// TIA Portal V17 export
// export: Created 2025-07-01T09:58:41.890921Z, ExportSetting WithDefaults, DisplayName Totally Integrated Automation Portal, DisplayVersion V17 Update 8, DisplayName TIA Portal Openness, DisplayVersion V17 Update 8, DisplayName TIA Portal Version Control Interface, DisplayVersion V17, DisplayName SINAMICS Startdrive Advanced, DisplayVersion V17 SP2, DisplayName SINAMICS Startdrive G110M, G120, G120C, G120D, G120P, G115D, DisplayVersion V17 SP2, DisplayName SINAMICS Startdrive G130, G150, S120, S150, SINAMICS MV, S210, DisplayVersion V17 SP2, DisplayName STEP 7 Professional, DisplayVersion V17 Update 8, DisplayName SINUMERIK ONE STEP 7 Toolbox, DisplayVersion V17 Update 12, DisplayName SINUMERIK ONE PLC Basic Program Plus, DisplayVersion V17 Update 12, DisplayName SINUMERIK 840D sl STEP 7 Toolbox, DisplayVersion V17 Update 12, DisplayName STEP 7 Safety, DisplayVersion V17 Update 6, DisplayName WinCC Advanced, DisplayVersion V17 Update 8
FUNCTION "FC442_MACHINE_RUN_OUT_ALARM_DECODING" : Void   // FC442, LAD
{ S7_Optimized_Access := 'FALSE' }
AUTHOR : ETXETAR
VERSION : 1.0
// stored: AutoNumber false, IsIECCheckEnabled false, SetENOAutomatically false, UDAEnableTagReadback false
   VAR_TEMP
      RST_ALARMS_1 : Bool;   // RESET ALARMS 1
      RST_ALARMS_2 : Bool;   // RESET ALARMS 2
      ZERO : Int;   // ZERO
      RET_VAL_1 : Int;   // RET VALUE
   END_VAR
   VAR CONSTANT
      FC_CONSTANT : Int := 440;
   END_VAR
   VAR_TEMP   // added for the SCL form of the ladder/FBD networks
      _w1 : Bool;
      _w2 : Bool;
      _w3 : Bool;
      _w4 : Bool;
      _w5 : Bool;
   END_VAR
BEGIN

REGION Network 1: ZERO
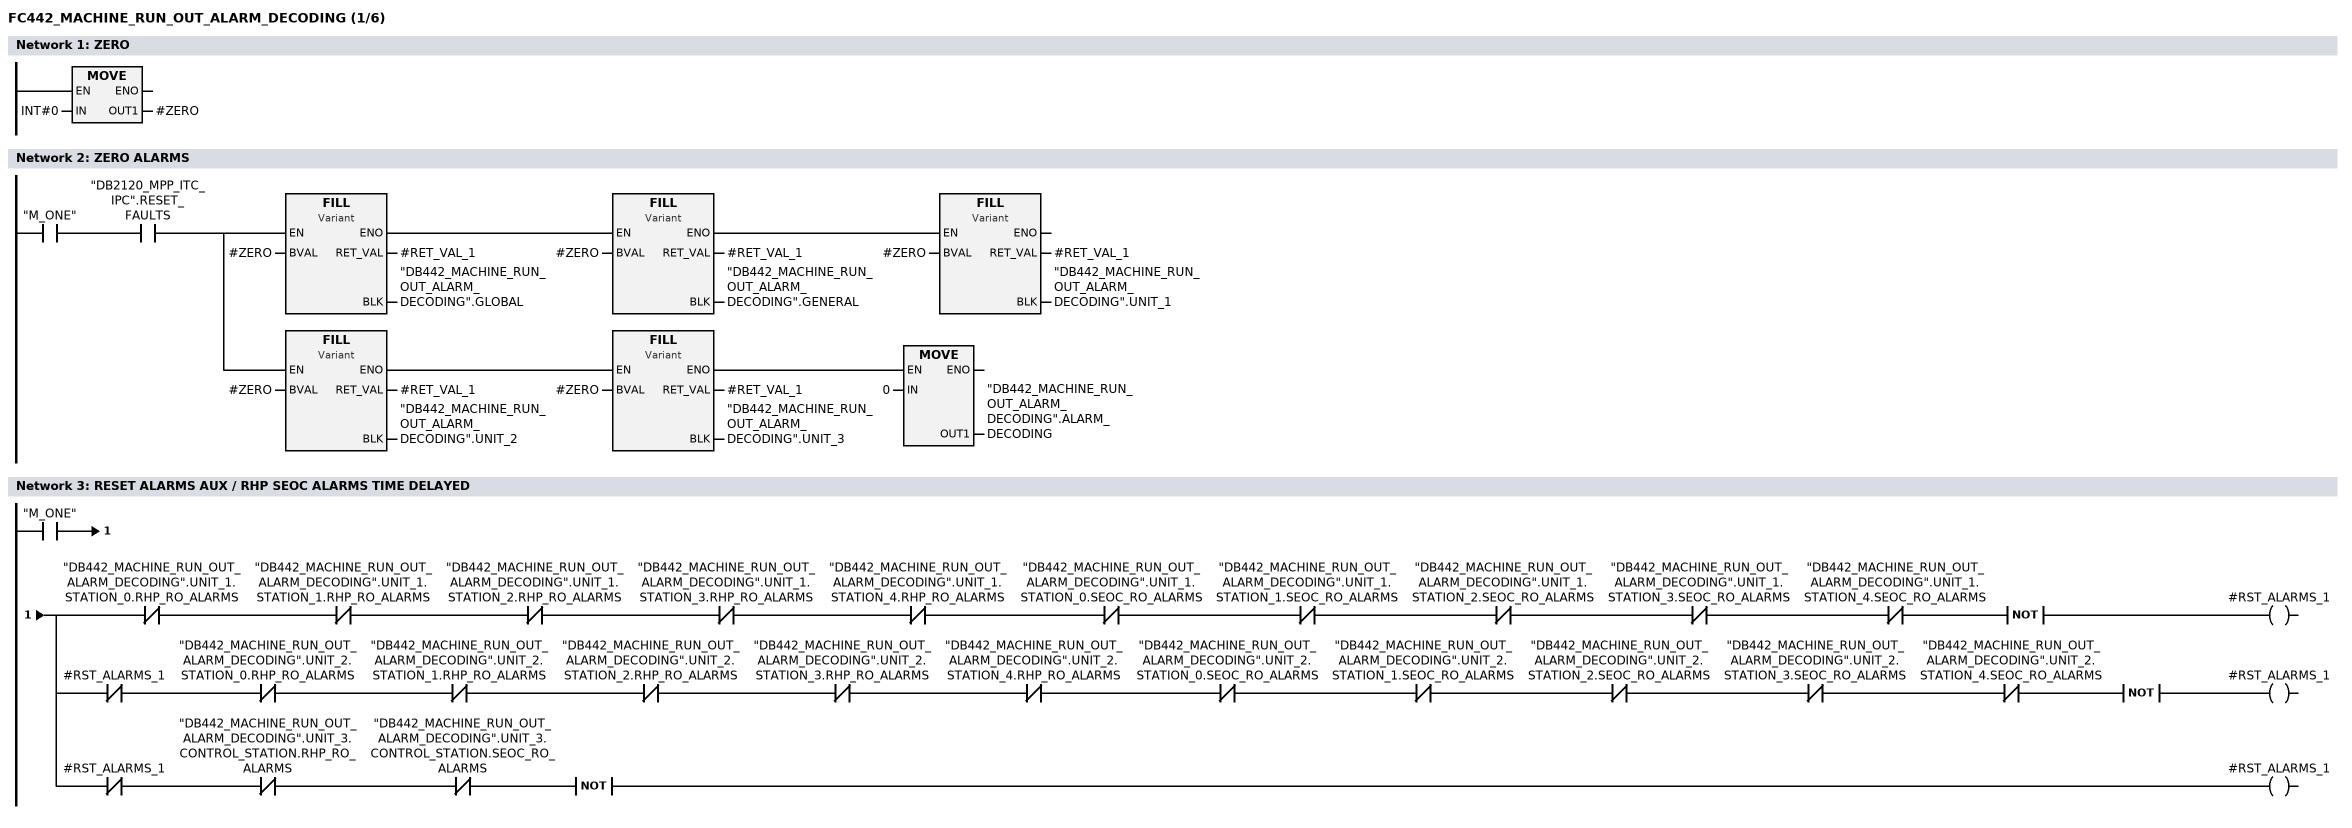
   RUNG wire#powerrail
      { S7_GenerateENO := "TRUE" } Move(in := INT#0, out1 => #ZERO)
   END_RUNG
   // the same network as SCL:
   #ZERO := INT#0;
END_REGION

REGION Network 2: ZERO ALARMS
   RUNG wire#powerrail
      Contact( "M_ONE" )
      Contact( "DB2120_MPP_ITC_IPC".RESET_FAULTS )
      wire#w1
      { S7_Templates := "ptr_type := Variant" } FILL(BVAL := #ZERO, RET_VAL => #RET_VAL_1, BLK => "DB442_MACHINE_RUN_OUT_ALARM_DECODING".GLOBAL)
      { S7_Templates := "ptr_type := Variant" } FILL(BVAL := #ZERO, RET_VAL => #RET_VAL_1, BLK => "DB442_MACHINE_RUN_OUT_ALARM_DECODING".GENERAL)
      { S7_Templates := "ptr_type := Variant" } FILL(BVAL := #ZERO, RET_VAL => #RET_VAL_1, BLK => "DB442_MACHINE_RUN_OUT_ALARM_DECODING".UNIT_1)
   END_RUNG
   RUNG wire#w1
      { S7_Templates := "ptr_type := Variant" } FILL(BVAL := #ZERO, RET_VAL => #RET_VAL_1, BLK => "DB442_MACHINE_RUN_OUT_ALARM_DECODING".UNIT_2)
      { S7_Templates := "ptr_type := Variant" } FILL(BVAL := #ZERO, RET_VAL => #RET_VAL_1, BLK => "DB442_MACHINE_RUN_OUT_ALARM_DECODING".UNIT_3)
      { S7_GenerateENO := "TRUE" } Move(in := 0, out1 => "DB442_MACHINE_RUN_OUT_ALARM_DECODING".ALARM_DECODING)
   END_RUNG
   // the same network as SCL:
   #_w2 := "M_ONE" AND "DB2120_MPP_ITC_IPC".RESET_FAULTS;
   #RET_VAL_1 := FILL(EN := "M_ONE" AND "DB2120_MPP_ITC_IPC".RESET_FAULTS,
                      BVAL := #ZERO,
                      BLK => "DB442_MACHINE_RUN_OUT_ALARM_DECODING".GLOBAL,
                      ENO => #_w1);
   #RET_VAL_1 := FILL(EN := #_w1,
                      BVAL := #ZERO,
                      BLK => "DB442_MACHINE_RUN_OUT_ALARM_DECODING".GENERAL,
                      ENO => #_w3);
   IF #_w3 THEN
       #RET_VAL_1 := FILL(BVAL := #ZERO, BLK => "DB442_MACHINE_RUN_OUT_ALARM_DECODING".UNIT_1);
   END_IF;
   #RET_VAL_1 := FILL(EN := #_w2,
                      BVAL := #ZERO,
                      BLK => "DB442_MACHINE_RUN_OUT_ALARM_DECODING".UNIT_2,
                      ENO => #_w4);
   #RET_VAL_1 := FILL(EN := #_w4,
                      BVAL := #ZERO,
                      BLK => "DB442_MACHINE_RUN_OUT_ALARM_DECODING".UNIT_3,
                      ENO => #_w5);
   IF #_w5 THEN "DB442_MACHINE_RUN_OUT_ALARM_DECODING".ALARM_DECODING := 0; END_IF;
END_REGION

REGION Network 3: RESET ALARMS AUX / RHP SEOC ALARMS TIME DELAYED
   RUNG wire#powerrail
      Contact( "M_ONE" )
      wire#w1
      I_Contact( "DB442_MACHINE_RUN_OUT_ALARM_DECODING".UNIT_1.STATION_0.RHP_RO_ALARMS )
      I_Contact( "DB442_MACHINE_RUN_OUT_ALARM_DECODING".UNIT_1.STATION_1.RHP_RO_ALARMS )
      I_Contact( "DB442_MACHINE_RUN_OUT_ALARM_DECODING".UNIT_1.STATION_2.RHP_RO_ALARMS )
      I_Contact( "DB442_MACHINE_RUN_OUT_ALARM_DECODING".UNIT_1.STATION_3.RHP_RO_ALARMS )
      I_Contact( "DB442_MACHINE_RUN_OUT_ALARM_DECODING".UNIT_1.STATION_4.RHP_RO_ALARMS )
      I_Contact( "DB442_MACHINE_RUN_OUT_ALARM_DECODING".UNIT_1.STATION_0.SEOC_RO_ALARMS )
      I_Contact( "DB442_MACHINE_RUN_OUT_ALARM_DECODING".UNIT_1.STATION_1.SEOC_RO_ALARMS )
      I_Contact( "DB442_MACHINE_RUN_OUT_ALARM_DECODING".UNIT_1.STATION_2.SEOC_RO_ALARMS )
      I_Contact( "DB442_MACHINE_RUN_OUT_ALARM_DECODING".UNIT_1.STATION_3.SEOC_RO_ALARMS )
      I_Contact( "DB442_MACHINE_RUN_OUT_ALARM_DECODING".UNIT_1.STATION_4.SEOC_RO_ALARMS )
      Not()
      Coil( #RST_ALARMS_1 )
   END_RUNG
   RUNG wire#w1
      I_Contact( #RST_ALARMS_1 )
      I_Contact( "DB442_MACHINE_RUN_OUT_ALARM_DECODING".UNIT_2.STATION_0.RHP_RO_ALARMS )
      I_Contact( "DB442_MACHINE_RUN_OUT_ALARM_DECODING".UNIT_2.STATION_1.RHP_RO_ALARMS )
      I_Contact( "DB442_MACHINE_RUN_OUT_ALARM_DECODING".UNIT_2.STATION_2.RHP_RO_ALARMS )
      I_Contact( "DB442_MACHINE_RUN_OUT_ALARM_DECODING".UNIT_2.STATION_3.RHP_RO_ALARMS )
      I_Contact( "DB442_MACHINE_RUN_OUT_ALARM_DECODING".UNIT_2.STATION_4.RHP_RO_ALARMS )
      I_Contact( "DB442_MACHINE_RUN_OUT_ALARM_DECODING".UNIT_2.STATION_0.SEOC_RO_ALARMS )
      I_Contact( "DB442_MACHINE_RUN_OUT_ALARM_DECODING".UNIT_2.STATION_1.SEOC_RO_ALARMS )
      I_Contact( "DB442_MACHINE_RUN_OUT_ALARM_DECODING".UNIT_2.STATION_2.SEOC_RO_ALARMS )
      I_Contact( "DB442_MACHINE_RUN_OUT_ALARM_DECODING".UNIT_2.STATION_3.SEOC_RO_ALARMS )
      I_Contact( "DB442_MACHINE_RUN_OUT_ALARM_DECODING".UNIT_2.STATION_4.SEOC_RO_ALARMS )
      Not()
      Coil( #RST_ALARMS_1 )
   END_RUNG
   RUNG wire#w1
      I_Contact( #RST_ALARMS_1 )
      I_Contact( "DB442_MACHINE_RUN_OUT_ALARM_DECODING".UNIT_3.CONTROL_STATION.RHP_RO_ALARMS )
      I_Contact( "DB442_MACHINE_RUN_OUT_ALARM_DECODING".UNIT_3.CONTROL_STATION.SEOC_RO_ALARMS )
      Not()
      Coil( #RST_ALARMS_1 )
   END_RUNG
   // the same network as SCL:
   #RST_ALARMS_1 := NOT ("M_ONE" AND NOT "DB442_MACHINE_RUN_OUT_ALARM_DECODING".UNIT_1.STATION_0.RHP_RO_ALARMS AND NOT "DB442_MACHINE_RUN_OUT_ALARM_DECODING".UNIT_1.STATION_1.RHP_RO_ALARMS AND NOT "DB442_MACHINE_RUN_OUT_ALARM_DECODING".UNIT_1.STATION_2.RHP_RO_ALARMS AND NOT "DB442_MACHINE_RUN_OUT_ALARM_DECODING".UNIT_1.STATION_3.RHP_RO_ALARMS AND NOT "DB442_MACHINE_RUN_OUT_ALARM_DECODING".UNIT_1.STATION_4.RHP_RO_ALARMS AND NOT "DB442_MACHINE_RUN_OUT_ALARM_DECODING".UNIT_1.STATION_0.SEOC_RO_ALARMS AND NOT "DB442_MACHINE_RUN_OUT_ALARM_DECODING".UNIT_1.STATION_1.SEOC_RO_ALARMS AND NOT "DB442_MACHINE_RUN_OUT_ALARM_DECODING".UNIT_1.STATION_2.SEOC_RO_ALARMS AND NOT "DB442_MACHINE_RUN_OUT_ALARM_DECODING".UNIT_1.STATION_3.SEOC_RO_ALARMS AND NOT "DB442_MACHINE_RUN_OUT_ALARM_DECODING".UNIT_1.STATION_4.SEOC_RO_ALARMS);
   #RST_ALARMS_1 := NOT ("M_ONE" AND NOT #RST_ALARMS_1 AND NOT "DB442_MACHINE_RUN_OUT_ALARM_DECODING".UNIT_2.STATION_0.RHP_RO_ALARMS AND NOT "DB442_MACHINE_RUN_OUT_ALARM_DECODING".UNIT_2.STATION_1.RHP_RO_ALARMS AND NOT "DB442_MACHINE_RUN_OUT_ALARM_DECODING".UNIT_2.STATION_2.RHP_RO_ALARMS AND NOT "DB442_MACHINE_RUN_OUT_ALARM_DECODING".UNIT_2.STATION_3.RHP_RO_ALARMS AND NOT "DB442_MACHINE_RUN_OUT_ALARM_DECODING".UNIT_2.STATION_4.RHP_RO_ALARMS AND NOT "DB442_MACHINE_RUN_OUT_ALARM_DECODING".UNIT_2.STATION_0.SEOC_RO_ALARMS AND NOT "DB442_MACHINE_RUN_OUT_ALARM_DECODING".UNIT_2.STATION_1.SEOC_RO_ALARMS AND NOT "DB442_MACHINE_RUN_OUT_ALARM_DECODING".UNIT_2.STATION_2.SEOC_RO_ALARMS AND NOT "DB442_MACHINE_RUN_OUT_ALARM_DECODING".UNIT_2.STATION_3.SEOC_RO_ALARMS AND NOT "DB442_MACHINE_RUN_OUT_ALARM_DECODING".UNIT_2.STATION_4.SEOC_RO_ALARMS);
   #RST_ALARMS_1 := NOT ("M_ONE" AND NOT #RST_ALARMS_1 AND NOT "DB442_MACHINE_RUN_OUT_ALARM_DECODING".UNIT_3.CONTROL_STATION.RHP_RO_ALARMS AND NOT "DB442_MACHINE_RUN_OUT_ALARM_DECODING".UNIT_3.CONTROL_STATION.SEOC_RO_ALARMS);
END_REGION

REGION Network 4: STATIONS ALARMS RESET / RETURN HOME POSITION & STOP END OF CYCLE ALARMS
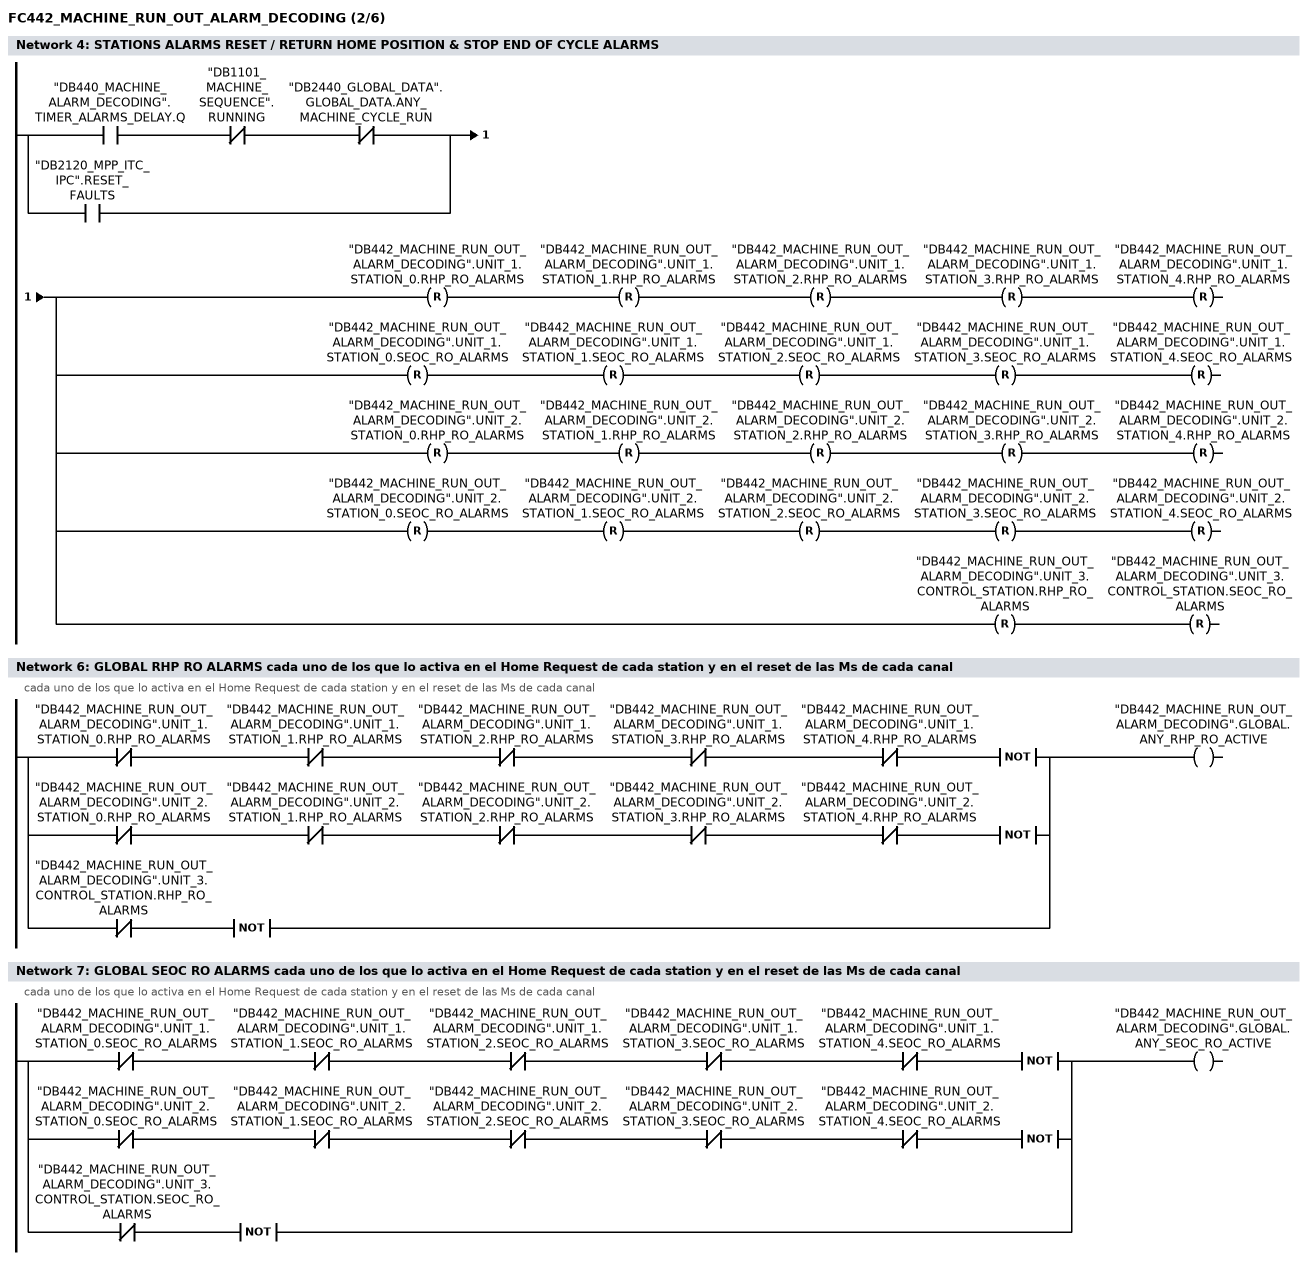
   RUNG wire#powerrail
      Contact( "DB440_MACHINE_ALARM_DECODING".TIMER_ALARMS_DELAY.Q )
      I_Contact( "DB1101_MACHINE_SEQUENCE".RUNNING )
      I_Contact( "DB2440_GLOBAL_DATA".GLOBAL_DATA.ANY_MACHINE_CYCLE_RUN )
      wire#w1
      R_Coil( "DB442_MACHINE_RUN_OUT_ALARM_DECODING".UNIT_1.STATION_0.RHP_RO_ALARMS )
      R_Coil( "DB442_MACHINE_RUN_OUT_ALARM_DECODING".UNIT_1.STATION_1.RHP_RO_ALARMS )
      R_Coil( "DB442_MACHINE_RUN_OUT_ALARM_DECODING".UNIT_1.STATION_2.RHP_RO_ALARMS )
      R_Coil( "DB442_MACHINE_RUN_OUT_ALARM_DECODING".UNIT_1.STATION_3.RHP_RO_ALARMS )
      R_Coil( "DB442_MACHINE_RUN_OUT_ALARM_DECODING".UNIT_1.STATION_4.RHP_RO_ALARMS )
   END_RUNG
   RUNG wire#powerrail
      Contact( "DB2120_MPP_ITC_IPC".RESET_FAULTS )
   END_RUNG wire#w1
   RUNG wire#w1
      R_Coil( "DB442_MACHINE_RUN_OUT_ALARM_DECODING".UNIT_1.STATION_0.SEOC_RO_ALARMS )
      R_Coil( "DB442_MACHINE_RUN_OUT_ALARM_DECODING".UNIT_1.STATION_1.SEOC_RO_ALARMS )
      R_Coil( "DB442_MACHINE_RUN_OUT_ALARM_DECODING".UNIT_1.STATION_2.SEOC_RO_ALARMS )
      R_Coil( "DB442_MACHINE_RUN_OUT_ALARM_DECODING".UNIT_1.STATION_3.SEOC_RO_ALARMS )
      R_Coil( "DB442_MACHINE_RUN_OUT_ALARM_DECODING".UNIT_1.STATION_4.SEOC_RO_ALARMS )
   END_RUNG
   RUNG wire#w1
      R_Coil( "DB442_MACHINE_RUN_OUT_ALARM_DECODING".UNIT_2.STATION_0.RHP_RO_ALARMS )
      R_Coil( "DB442_MACHINE_RUN_OUT_ALARM_DECODING".UNIT_2.STATION_1.RHP_RO_ALARMS )
      R_Coil( "DB442_MACHINE_RUN_OUT_ALARM_DECODING".UNIT_2.STATION_2.RHP_RO_ALARMS )
      R_Coil( "DB442_MACHINE_RUN_OUT_ALARM_DECODING".UNIT_2.STATION_3.RHP_RO_ALARMS )
      R_Coil( "DB442_MACHINE_RUN_OUT_ALARM_DECODING".UNIT_2.STATION_4.RHP_RO_ALARMS )
   END_RUNG
   RUNG wire#w1
      R_Coil( "DB442_MACHINE_RUN_OUT_ALARM_DECODING".UNIT_2.STATION_0.SEOC_RO_ALARMS )
      R_Coil( "DB442_MACHINE_RUN_OUT_ALARM_DECODING".UNIT_2.STATION_1.SEOC_RO_ALARMS )
      R_Coil( "DB442_MACHINE_RUN_OUT_ALARM_DECODING".UNIT_2.STATION_2.SEOC_RO_ALARMS )
      R_Coil( "DB442_MACHINE_RUN_OUT_ALARM_DECODING".UNIT_2.STATION_3.SEOC_RO_ALARMS )
      R_Coil( "DB442_MACHINE_RUN_OUT_ALARM_DECODING".UNIT_2.STATION_4.SEOC_RO_ALARMS )
   END_RUNG
   RUNG wire#w1
      R_Coil( "DB442_MACHINE_RUN_OUT_ALARM_DECODING".UNIT_3.CONTROL_STATION.RHP_RO_ALARMS )
      R_Coil( "DB442_MACHINE_RUN_OUT_ALARM_DECODING".UNIT_3.CONTROL_STATION.SEOC_RO_ALARMS )
   END_RUNG
   // the same network as SCL:
   IF ("DB440_MACHINE_ALARM_DECODING".TIMER_ALARMS_DELAY.Q AND NOT "DB1101_MACHINE_SEQUENCE".RUNNING AND NOT "DB2440_GLOBAL_DATA".GLOBAL_DATA.ANY_MACHINE_CYCLE_RUN) OR "DB2120_MPP_ITC_IPC".RESET_FAULTS THEN
       "DB442_MACHINE_RUN_OUT_ALARM_DECODING".UNIT_1.STATION_0.RHP_RO_ALARMS := FALSE;
       "DB442_MACHINE_RUN_OUT_ALARM_DECODING".UNIT_1.STATION_1.RHP_RO_ALARMS := FALSE;
       "DB442_MACHINE_RUN_OUT_ALARM_DECODING".UNIT_1.STATION_2.RHP_RO_ALARMS := FALSE;
       "DB442_MACHINE_RUN_OUT_ALARM_DECODING".UNIT_1.STATION_3.RHP_RO_ALARMS := FALSE;
       "DB442_MACHINE_RUN_OUT_ALARM_DECODING".UNIT_1.STATION_4.RHP_RO_ALARMS := FALSE;
       "DB442_MACHINE_RUN_OUT_ALARM_DECODING".UNIT_1.STATION_0.SEOC_RO_ALARMS := FALSE;
       "DB442_MACHINE_RUN_OUT_ALARM_DECODING".UNIT_1.STATION_1.SEOC_RO_ALARMS := FALSE;
       "DB442_MACHINE_RUN_OUT_ALARM_DECODING".UNIT_1.STATION_2.SEOC_RO_ALARMS := FALSE;
       "DB442_MACHINE_RUN_OUT_ALARM_DECODING".UNIT_1.STATION_3.SEOC_RO_ALARMS := FALSE;
       "DB442_MACHINE_RUN_OUT_ALARM_DECODING".UNIT_1.STATION_4.SEOC_RO_ALARMS := FALSE;
       "DB442_MACHINE_RUN_OUT_ALARM_DECODING".UNIT_2.STATION_0.RHP_RO_ALARMS := FALSE;
       "DB442_MACHINE_RUN_OUT_ALARM_DECODING".UNIT_2.STATION_1.RHP_RO_ALARMS := FALSE;
       "DB442_MACHINE_RUN_OUT_ALARM_DECODING".UNIT_2.STATION_2.RHP_RO_ALARMS := FALSE;
       "DB442_MACHINE_RUN_OUT_ALARM_DECODING".UNIT_2.STATION_3.RHP_RO_ALARMS := FALSE;
       "DB442_MACHINE_RUN_OUT_ALARM_DECODING".UNIT_2.STATION_4.RHP_RO_ALARMS := FALSE;
       "DB442_MACHINE_RUN_OUT_ALARM_DECODING".UNIT_2.STATION_0.SEOC_RO_ALARMS := FALSE;
       "DB442_MACHINE_RUN_OUT_ALARM_DECODING".UNIT_2.STATION_1.SEOC_RO_ALARMS := FALSE;
       "DB442_MACHINE_RUN_OUT_ALARM_DECODING".UNIT_2.STATION_2.SEOC_RO_ALARMS := FALSE;
       "DB442_MACHINE_RUN_OUT_ALARM_DECODING".UNIT_2.STATION_3.SEOC_RO_ALARMS := FALSE;
       "DB442_MACHINE_RUN_OUT_ALARM_DECODING".UNIT_2.STATION_4.SEOC_RO_ALARMS := FALSE;
       "DB442_MACHINE_RUN_OUT_ALARM_DECODING".UNIT_3.CONTROL_STATION.RHP_RO_ALARMS := FALSE;
       "DB442_MACHINE_RUN_OUT_ALARM_DECODING".UNIT_3.CONTROL_STATION.SEOC_RO_ALARMS := FALSE;
   END_IF;
END_REGION

REGION Network 5: <<<<<<<<<<<<<<<<<<<< ALARMS GLOBAL>>>>>>>>>>>>>>>>>>>>
END_REGION

REGION Network 6: GLOBAL RHP RO ALARMS cada uno de los que lo activa en el Home Request de cada station y en el reset de las Ms de cada canal
   // cada uno de los que lo activa en el Home Request de cada station y en el reset de las Ms de cada canal
   RUNG wire#powerrail
      I_Contact( "DB442_MACHINE_RUN_OUT_ALARM_DECODING".UNIT_1.STATION_0.RHP_RO_ALARMS )
      I_Contact( "DB442_MACHINE_RUN_OUT_ALARM_DECODING".UNIT_1.STATION_1.RHP_RO_ALARMS )
      I_Contact( "DB442_MACHINE_RUN_OUT_ALARM_DECODING".UNIT_1.STATION_2.RHP_RO_ALARMS )
      I_Contact( "DB442_MACHINE_RUN_OUT_ALARM_DECODING".UNIT_1.STATION_3.RHP_RO_ALARMS )
      I_Contact( "DB442_MACHINE_RUN_OUT_ALARM_DECODING".UNIT_1.STATION_4.RHP_RO_ALARMS )
      Not()
      wire#w1
      Coil( "DB442_MACHINE_RUN_OUT_ALARM_DECODING".GLOBAL.ANY_RHP_RO_ACTIVE )
   END_RUNG
   RUNG wire#powerrail
      I_Contact( "DB442_MACHINE_RUN_OUT_ALARM_DECODING".UNIT_2.STATION_0.RHP_RO_ALARMS )
      I_Contact( "DB442_MACHINE_RUN_OUT_ALARM_DECODING".UNIT_2.STATION_1.RHP_RO_ALARMS )
      I_Contact( "DB442_MACHINE_RUN_OUT_ALARM_DECODING".UNIT_2.STATION_2.RHP_RO_ALARMS )
      I_Contact( "DB442_MACHINE_RUN_OUT_ALARM_DECODING".UNIT_2.STATION_3.RHP_RO_ALARMS )
      I_Contact( "DB442_MACHINE_RUN_OUT_ALARM_DECODING".UNIT_2.STATION_4.RHP_RO_ALARMS )
      Not()
   END_RUNG wire#w1
   RUNG wire#powerrail
      I_Contact( "DB442_MACHINE_RUN_OUT_ALARM_DECODING".UNIT_3.CONTROL_STATION.RHP_RO_ALARMS )
      Not()
   END_RUNG wire#w1
   // the same network as SCL:
   "DB442_MACHINE_RUN_OUT_ALARM_DECODING".GLOBAL.ANY_RHP_RO_ACTIVE := NOT (NOT "DB442_MACHINE_RUN_OUT_ALARM_DECODING".UNIT_1.STATION_0.RHP_RO_ALARMS AND NOT "DB442_MACHINE_RUN_OUT_ALARM_DECODING".UNIT_1.STATION_1.RHP_RO_ALARMS AND NOT "DB442_MACHINE_RUN_OUT_ALARM_DECODING".UNIT_1.STATION_2.RHP_RO_ALARMS AND NOT "DB442_MACHINE_RUN_OUT_ALARM_DECODING".UNIT_1.STATION_3.RHP_RO_ALARMS AND NOT "DB442_MACHINE_RUN_OUT_ALARM_DECODING".UNIT_1.STATION_4.RHP_RO_ALARMS) OR NOT (NOT "DB442_MACHINE_RUN_OUT_ALARM_DECODING".UNIT_2.STATION_0.RHP_RO_ALARMS AND NOT "DB442_MACHINE_RUN_OUT_ALARM_DECODING".UNIT_2.STATION_1.RHP_RO_ALARMS AND NOT "DB442_MACHINE_RUN_OUT_ALARM_DECODING".UNIT_2.STATION_2.RHP_RO_ALARMS AND NOT "DB442_MACHINE_RUN_OUT_ALARM_DECODING".UNIT_2.STATION_3.RHP_RO_ALARMS AND NOT "DB442_MACHINE_RUN_OUT_ALARM_DECODING".UNIT_2.STATION_4.RHP_RO_ALARMS) OR NOT (NOT "DB442_MACHINE_RUN_OUT_ALARM_DECODING".UNIT_3.CONTROL_STATION.RHP_RO_ALARMS);
END_REGION

REGION Network 7: GLOBAL SEOC RO ALARMS cada uno de los que lo activa en el Home Request de cada station y en el reset de las Ms de cada canal
   // cada uno de los que lo activa en el Home Request de cada station y en el reset de las Ms de cada canal
   RUNG wire#powerrail
      I_Contact( "DB442_MACHINE_RUN_OUT_ALARM_DECODING".UNIT_1.STATION_0.SEOC_RO_ALARMS )
      I_Contact( "DB442_MACHINE_RUN_OUT_ALARM_DECODING".UNIT_1.STATION_1.SEOC_RO_ALARMS )
      I_Contact( "DB442_MACHINE_RUN_OUT_ALARM_DECODING".UNIT_1.STATION_2.SEOC_RO_ALARMS )
      I_Contact( "DB442_MACHINE_RUN_OUT_ALARM_DECODING".UNIT_1.STATION_3.SEOC_RO_ALARMS )
      I_Contact( "DB442_MACHINE_RUN_OUT_ALARM_DECODING".UNIT_1.STATION_4.SEOC_RO_ALARMS )
      Not()
      wire#w1
      Coil( "DB442_MACHINE_RUN_OUT_ALARM_DECODING".GLOBAL.ANY_SEOC_RO_ACTIVE )
   END_RUNG
   RUNG wire#powerrail
      I_Contact( "DB442_MACHINE_RUN_OUT_ALARM_DECODING".UNIT_2.STATION_0.SEOC_RO_ALARMS )
      I_Contact( "DB442_MACHINE_RUN_OUT_ALARM_DECODING".UNIT_2.STATION_1.SEOC_RO_ALARMS )
      I_Contact( "DB442_MACHINE_RUN_OUT_ALARM_DECODING".UNIT_2.STATION_2.SEOC_RO_ALARMS )
      I_Contact( "DB442_MACHINE_RUN_OUT_ALARM_DECODING".UNIT_2.STATION_3.SEOC_RO_ALARMS )
      I_Contact( "DB442_MACHINE_RUN_OUT_ALARM_DECODING".UNIT_2.STATION_4.SEOC_RO_ALARMS )
      Not()
   END_RUNG wire#w1
   RUNG wire#powerrail
      I_Contact( "DB442_MACHINE_RUN_OUT_ALARM_DECODING".UNIT_3.CONTROL_STATION.SEOC_RO_ALARMS )
      Not()
   END_RUNG wire#w1
   // the same network as SCL:
   "DB442_MACHINE_RUN_OUT_ALARM_DECODING".GLOBAL.ANY_SEOC_RO_ACTIVE := NOT (NOT "DB442_MACHINE_RUN_OUT_ALARM_DECODING".UNIT_1.STATION_0.SEOC_RO_ALARMS AND NOT "DB442_MACHINE_RUN_OUT_ALARM_DECODING".UNIT_1.STATION_1.SEOC_RO_ALARMS AND NOT "DB442_MACHINE_RUN_OUT_ALARM_DECODING".UNIT_1.STATION_2.SEOC_RO_ALARMS AND NOT "DB442_MACHINE_RUN_OUT_ALARM_DECODING".UNIT_1.STATION_3.SEOC_RO_ALARMS AND NOT "DB442_MACHINE_RUN_OUT_ALARM_DECODING".UNIT_1.STATION_4.SEOC_RO_ALARMS) OR NOT (NOT "DB442_MACHINE_RUN_OUT_ALARM_DECODING".UNIT_2.STATION_0.SEOC_RO_ALARMS AND NOT "DB442_MACHINE_RUN_OUT_ALARM_DECODING".UNIT_2.STATION_1.SEOC_RO_ALARMS AND NOT "DB442_MACHINE_RUN_OUT_ALARM_DECODING".UNIT_2.STATION_2.SEOC_RO_ALARMS AND NOT "DB442_MACHINE_RUN_OUT_ALARM_DECODING".UNIT_2.STATION_3.SEOC_RO_ALARMS AND NOT "DB442_MACHINE_RUN_OUT_ALARM_DECODING".UNIT_2.STATION_4.SEOC_RO_ALARMS) OR NOT (NOT "DB442_MACHINE_RUN_OUT_ALARM_DECODING".UNIT_3.CONTROL_STATION.SEOC_RO_ALARMS);
END_REGION

REGION Network 8: GLOBAL ANY RUN OUT ALARM ACTIVE (esta iría en el run out request)
   // (esta iría en el run out request)
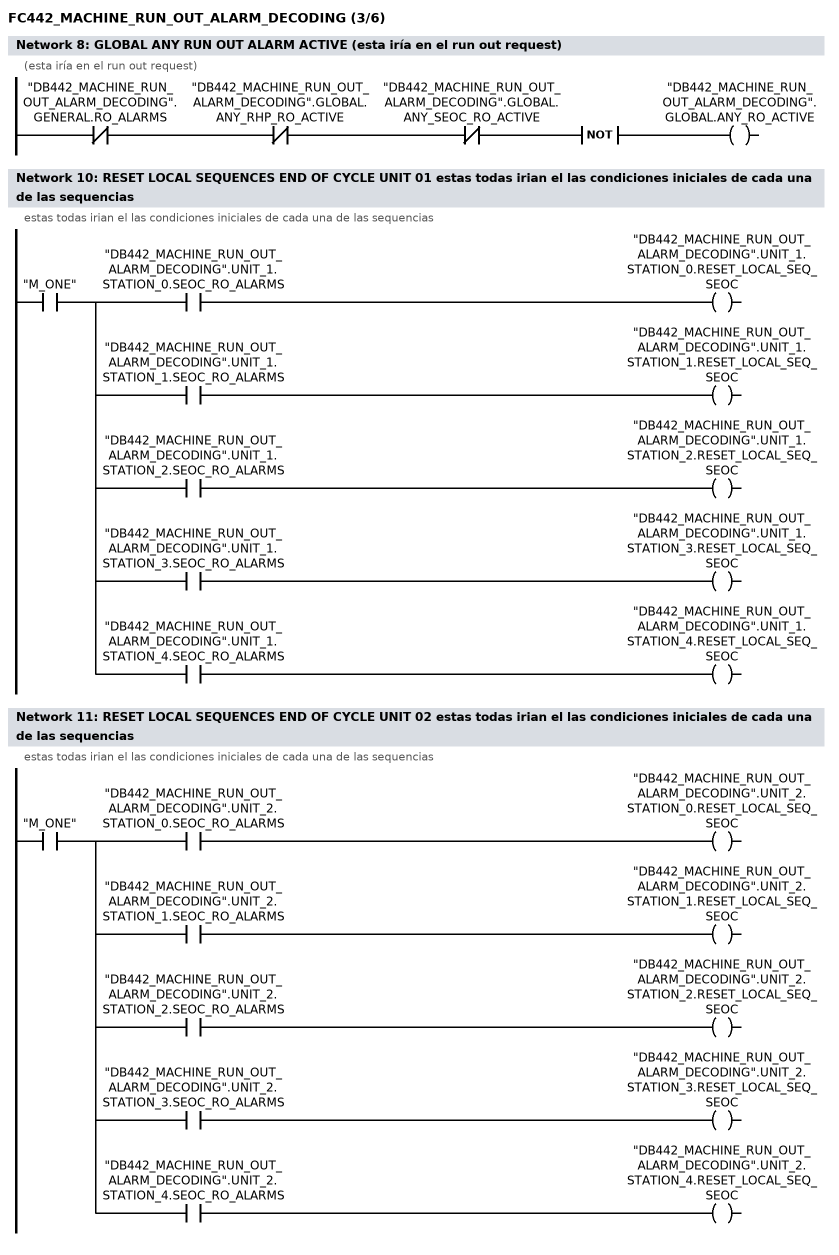
   RUNG wire#powerrail
      I_Contact( "DB442_MACHINE_RUN_OUT_ALARM_DECODING".GENERAL.RO_ALARMS )
      I_Contact( "DB442_MACHINE_RUN_OUT_ALARM_DECODING".GLOBAL.ANY_RHP_RO_ACTIVE )
      I_Contact( "DB442_MACHINE_RUN_OUT_ALARM_DECODING".GLOBAL.ANY_SEOC_RO_ACTIVE )
      Not()
      Coil( "DB442_MACHINE_RUN_OUT_ALARM_DECODING".GLOBAL.ANY_RO_ACTIVE )
   END_RUNG
   // the same network as SCL:
   "DB442_MACHINE_RUN_OUT_ALARM_DECODING".GLOBAL.ANY_RO_ACTIVE := NOT (NOT "DB442_MACHINE_RUN_OUT_ALARM_DECODING".GENERAL.RO_ALARMS AND NOT "DB442_MACHINE_RUN_OUT_ALARM_DECODING".GLOBAL.ANY_RHP_RO_ACTIVE AND NOT "DB442_MACHINE_RUN_OUT_ALARM_DECODING".GLOBAL.ANY_SEOC_RO_ACTIVE);
END_REGION

REGION Network 9: <<<<<<<<<<<<<<<<<<<< RESET LOCAL SEQUENCES >>>>>>>>>>>>>>>>>>>>
END_REGION

REGION Network 10: RESET LOCAL SEQUENCES END OF CYCLE UNIT 01 estas todas irian el las condiciones iniciales de cada una de las sequencias
   // estas todas irian el las condiciones iniciales de cada una de las sequencias
   RUNG wire#powerrail
      Contact( "M_ONE" )
      wire#w1
      Contact( "DB442_MACHINE_RUN_OUT_ALARM_DECODING".UNIT_1.STATION_0.SEOC_RO_ALARMS )
      Coil( "DB442_MACHINE_RUN_OUT_ALARM_DECODING".UNIT_1.STATION_0.RESET_LOCAL_SEQ_SEOC )
   END_RUNG
   RUNG wire#w1
      Contact( "DB442_MACHINE_RUN_OUT_ALARM_DECODING".UNIT_1.STATION_1.SEOC_RO_ALARMS )
      Coil( "DB442_MACHINE_RUN_OUT_ALARM_DECODING".UNIT_1.STATION_1.RESET_LOCAL_SEQ_SEOC )
   END_RUNG
   RUNG wire#w1
      Contact( "DB442_MACHINE_RUN_OUT_ALARM_DECODING".UNIT_1.STATION_2.SEOC_RO_ALARMS )
      Coil( "DB442_MACHINE_RUN_OUT_ALARM_DECODING".UNIT_1.STATION_2.RESET_LOCAL_SEQ_SEOC )
   END_RUNG
   RUNG wire#w1
      Contact( "DB442_MACHINE_RUN_OUT_ALARM_DECODING".UNIT_1.STATION_3.SEOC_RO_ALARMS )
      Coil( "DB442_MACHINE_RUN_OUT_ALARM_DECODING".UNIT_1.STATION_3.RESET_LOCAL_SEQ_SEOC )
   END_RUNG
   RUNG wire#w1
      Contact( "DB442_MACHINE_RUN_OUT_ALARM_DECODING".UNIT_1.STATION_4.SEOC_RO_ALARMS )
      Coil( "DB442_MACHINE_RUN_OUT_ALARM_DECODING".UNIT_1.STATION_4.RESET_LOCAL_SEQ_SEOC )
   END_RUNG
   // the same network as SCL:
   "DB442_MACHINE_RUN_OUT_ALARM_DECODING".UNIT_1.STATION_0.RESET_LOCAL_SEQ_SEOC := "M_ONE" AND "DB442_MACHINE_RUN_OUT_ALARM_DECODING".UNIT_1.STATION_0.SEOC_RO_ALARMS;
   "DB442_MACHINE_RUN_OUT_ALARM_DECODING".UNIT_1.STATION_1.RESET_LOCAL_SEQ_SEOC := "M_ONE" AND "DB442_MACHINE_RUN_OUT_ALARM_DECODING".UNIT_1.STATION_1.SEOC_RO_ALARMS;
   "DB442_MACHINE_RUN_OUT_ALARM_DECODING".UNIT_1.STATION_2.RESET_LOCAL_SEQ_SEOC := "M_ONE" AND "DB442_MACHINE_RUN_OUT_ALARM_DECODING".UNIT_1.STATION_2.SEOC_RO_ALARMS;
   "DB442_MACHINE_RUN_OUT_ALARM_DECODING".UNIT_1.STATION_3.RESET_LOCAL_SEQ_SEOC := "M_ONE" AND "DB442_MACHINE_RUN_OUT_ALARM_DECODING".UNIT_1.STATION_3.SEOC_RO_ALARMS;
   "DB442_MACHINE_RUN_OUT_ALARM_DECODING".UNIT_1.STATION_4.RESET_LOCAL_SEQ_SEOC := "M_ONE" AND "DB442_MACHINE_RUN_OUT_ALARM_DECODING".UNIT_1.STATION_4.SEOC_RO_ALARMS;
END_REGION

REGION Network 11: RESET LOCAL SEQUENCES END OF CYCLE UNIT 02 estas todas irian el las condiciones iniciales de cada una de las sequencias
   // estas todas irian el las condiciones iniciales de cada una de las sequencias
   RUNG wire#powerrail
      Contact( "M_ONE" )
      wire#w1
      Contact( "DB442_MACHINE_RUN_OUT_ALARM_DECODING".UNIT_2.STATION_0.SEOC_RO_ALARMS )
      Coil( "DB442_MACHINE_RUN_OUT_ALARM_DECODING".UNIT_2.STATION_0.RESET_LOCAL_SEQ_SEOC )
   END_RUNG
   RUNG wire#w1
      Contact( "DB442_MACHINE_RUN_OUT_ALARM_DECODING".UNIT_2.STATION_1.SEOC_RO_ALARMS )
      Coil( "DB442_MACHINE_RUN_OUT_ALARM_DECODING".UNIT_2.STATION_1.RESET_LOCAL_SEQ_SEOC )
   END_RUNG
   RUNG wire#w1
      Contact( "DB442_MACHINE_RUN_OUT_ALARM_DECODING".UNIT_2.STATION_2.SEOC_RO_ALARMS )
      Coil( "DB442_MACHINE_RUN_OUT_ALARM_DECODING".UNIT_2.STATION_2.RESET_LOCAL_SEQ_SEOC )
   END_RUNG
   RUNG wire#w1
      Contact( "DB442_MACHINE_RUN_OUT_ALARM_DECODING".UNIT_2.STATION_3.SEOC_RO_ALARMS )
      Coil( "DB442_MACHINE_RUN_OUT_ALARM_DECODING".UNIT_2.STATION_3.RESET_LOCAL_SEQ_SEOC )
   END_RUNG
   RUNG wire#w1
      Contact( "DB442_MACHINE_RUN_OUT_ALARM_DECODING".UNIT_2.STATION_4.SEOC_RO_ALARMS )
      Coil( "DB442_MACHINE_RUN_OUT_ALARM_DECODING".UNIT_2.STATION_4.RESET_LOCAL_SEQ_SEOC )
   END_RUNG
   // the same network as SCL:
   "DB442_MACHINE_RUN_OUT_ALARM_DECODING".UNIT_2.STATION_0.RESET_LOCAL_SEQ_SEOC := "M_ONE" AND "DB442_MACHINE_RUN_OUT_ALARM_DECODING".UNIT_2.STATION_0.SEOC_RO_ALARMS;
   "DB442_MACHINE_RUN_OUT_ALARM_DECODING".UNIT_2.STATION_1.RESET_LOCAL_SEQ_SEOC := "M_ONE" AND "DB442_MACHINE_RUN_OUT_ALARM_DECODING".UNIT_2.STATION_1.SEOC_RO_ALARMS;
   "DB442_MACHINE_RUN_OUT_ALARM_DECODING".UNIT_2.STATION_2.RESET_LOCAL_SEQ_SEOC := "M_ONE" AND "DB442_MACHINE_RUN_OUT_ALARM_DECODING".UNIT_2.STATION_2.SEOC_RO_ALARMS;
   "DB442_MACHINE_RUN_OUT_ALARM_DECODING".UNIT_2.STATION_3.RESET_LOCAL_SEQ_SEOC := "M_ONE" AND "DB442_MACHINE_RUN_OUT_ALARM_DECODING".UNIT_2.STATION_3.SEOC_RO_ALARMS;
   "DB442_MACHINE_RUN_OUT_ALARM_DECODING".UNIT_2.STATION_4.RESET_LOCAL_SEQ_SEOC := "M_ONE" AND "DB442_MACHINE_RUN_OUT_ALARM_DECODING".UNIT_2.STATION_4.SEOC_RO_ALARMS;
END_REGION

REGION Network 12: RESET LOCAL SEQUENCES END OF CYCLE UNIT 03 estas todas irian el las condiciones iniciales de cada una de las sequencias
   // estas todas irian el las condiciones iniciales de cada una de las sequencias
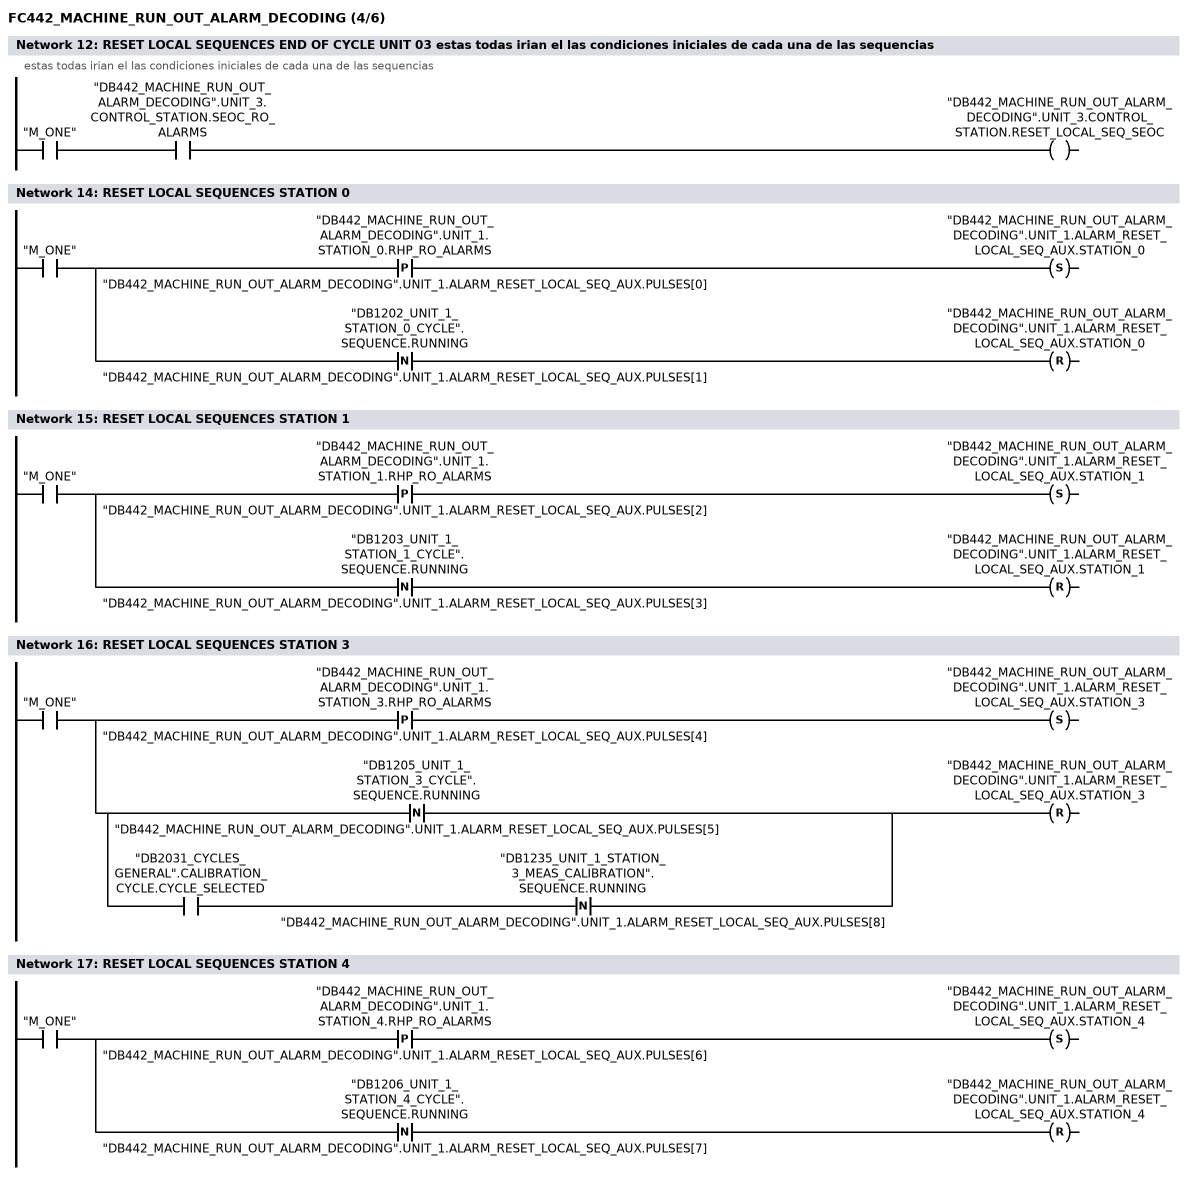
   RUNG wire#powerrail
      Contact( "M_ONE" )
      Contact( "DB442_MACHINE_RUN_OUT_ALARM_DECODING".UNIT_3.CONTROL_STATION.SEOC_RO_ALARMS )
      Coil( "DB442_MACHINE_RUN_OUT_ALARM_DECODING".UNIT_3.CONTROL_STATION.RESET_LOCAL_SEQ_SEOC )
   END_RUNG
   // the same network as SCL:
   "DB442_MACHINE_RUN_OUT_ALARM_DECODING".UNIT_3.CONTROL_STATION.RESET_LOCAL_SEQ_SEOC := "M_ONE" AND "DB442_MACHINE_RUN_OUT_ALARM_DECODING".UNIT_3.CONTROL_STATION.SEOC_RO_ALARMS;
END_REGION

REGION Network 13: <<<<<<<<<<<<<< RESET LOCAL SEQUENCES AUXILIAR UNIT 1 >>>>>>>>>>>>>>
END_REGION

REGION Network 14: RESET LOCAL SEQUENCES STATION 0
   RUNG wire#powerrail
      Contact( "M_ONE" )
      wire#w1
      P_Contact(operand := "DB442_MACHINE_RUN_OUT_ALARM_DECODING".UNIT_1.STATION_0.RHP_RO_ALARMS, bit := "DB442_MACHINE_RUN_OUT_ALARM_DECODING".UNIT_1.ALARM_RESET_LOCAL_SEQ_AUX.PULSES[0])
      S_Coil( "DB442_MACHINE_RUN_OUT_ALARM_DECODING".UNIT_1.ALARM_RESET_LOCAL_SEQ_AUX.STATION_0 )
   END_RUNG
   RUNG wire#w1
      N_Contact(operand := "DB1202_UNIT_1_STATION_0_CYCLE".SEQUENCE.RUNNING, bit := "DB442_MACHINE_RUN_OUT_ALARM_DECODING".UNIT_1.ALARM_RESET_LOCAL_SEQ_AUX.PULSES[1])
      R_Coil( "DB442_MACHINE_RUN_OUT_ALARM_DECODING".UNIT_1.ALARM_RESET_LOCAL_SEQ_AUX.STATION_0 )
   END_RUNG
   // the same network as SCL:
   #_w1 := "M_ONE" AND "DB442_MACHINE_RUN_OUT_ALARM_DECODING".UNIT_1.STATION_0.RHP_RO_ALARMS AND NOT "DB442_MACHINE_RUN_OUT_ALARM_DECODING".UNIT_1.ALARM_RESET_LOCAL_SEQ_AUX.PULSES[0];   // rising edge of "DB442_MACHINE_RUN_OUT_ALARM_DECODING".UNIT_1.STATION_0.RHP_RO_ALARMS
   "DB442_MACHINE_RUN_OUT_ALARM_DECODING".UNIT_1.ALARM_RESET_LOCAL_SEQ_AUX.PULSES[0] := "DB442_MACHINE_RUN_OUT_ALARM_DECODING".UNIT_1.STATION_0.RHP_RO_ALARMS;
   IF #_w1 THEN
       "DB442_MACHINE_RUN_OUT_ALARM_DECODING".UNIT_1.ALARM_RESET_LOCAL_SEQ_AUX.STATION_0 := TRUE;
   END_IF;
   #_w2 := "M_ONE" AND NOT "DB1202_UNIT_1_STATION_0_CYCLE".SEQUENCE.RUNNING AND "DB442_MACHINE_RUN_OUT_ALARM_DECODING".UNIT_1.ALARM_RESET_LOCAL_SEQ_AUX.PULSES[1];   // falling edge of "DB1202_UNIT_1_STATION_0_CYCLE".SEQUENCE.RUNNING
   "DB442_MACHINE_RUN_OUT_ALARM_DECODING".UNIT_1.ALARM_RESET_LOCAL_SEQ_AUX.PULSES[1] := "DB1202_UNIT_1_STATION_0_CYCLE".SEQUENCE.RUNNING;
   IF #_w2 THEN
       "DB442_MACHINE_RUN_OUT_ALARM_DECODING".UNIT_1.ALARM_RESET_LOCAL_SEQ_AUX.STATION_0 := FALSE;
   END_IF;
END_REGION

REGION Network 15: RESET LOCAL SEQUENCES STATION 1
   RUNG wire#powerrail
      Contact( "M_ONE" )
      wire#w1
      P_Contact(operand := "DB442_MACHINE_RUN_OUT_ALARM_DECODING".UNIT_1.STATION_1.RHP_RO_ALARMS, bit := "DB442_MACHINE_RUN_OUT_ALARM_DECODING".UNIT_1.ALARM_RESET_LOCAL_SEQ_AUX.PULSES[2])
      S_Coil( "DB442_MACHINE_RUN_OUT_ALARM_DECODING".UNIT_1.ALARM_RESET_LOCAL_SEQ_AUX.STATION_1 )
   END_RUNG
   RUNG wire#w1
      N_Contact(operand := "DB1203_UNIT_1_STATION_1_CYCLE".SEQUENCE.RUNNING, bit := "DB442_MACHINE_RUN_OUT_ALARM_DECODING".UNIT_1.ALARM_RESET_LOCAL_SEQ_AUX.PULSES[3])
      R_Coil( "DB442_MACHINE_RUN_OUT_ALARM_DECODING".UNIT_1.ALARM_RESET_LOCAL_SEQ_AUX.STATION_1 )
   END_RUNG
   // the same network as SCL:
   #_w1 := "M_ONE" AND "DB442_MACHINE_RUN_OUT_ALARM_DECODING".UNIT_1.STATION_1.RHP_RO_ALARMS AND NOT "DB442_MACHINE_RUN_OUT_ALARM_DECODING".UNIT_1.ALARM_RESET_LOCAL_SEQ_AUX.PULSES[2];   // rising edge of "DB442_MACHINE_RUN_OUT_ALARM_DECODING".UNIT_1.STATION_1.RHP_RO_ALARMS
   "DB442_MACHINE_RUN_OUT_ALARM_DECODING".UNIT_1.ALARM_RESET_LOCAL_SEQ_AUX.PULSES[2] := "DB442_MACHINE_RUN_OUT_ALARM_DECODING".UNIT_1.STATION_1.RHP_RO_ALARMS;
   IF #_w1 THEN
       "DB442_MACHINE_RUN_OUT_ALARM_DECODING".UNIT_1.ALARM_RESET_LOCAL_SEQ_AUX.STATION_1 := TRUE;
   END_IF;
   #_w2 := "M_ONE" AND NOT "DB1203_UNIT_1_STATION_1_CYCLE".SEQUENCE.RUNNING AND "DB442_MACHINE_RUN_OUT_ALARM_DECODING".UNIT_1.ALARM_RESET_LOCAL_SEQ_AUX.PULSES[3];   // falling edge of "DB1203_UNIT_1_STATION_1_CYCLE".SEQUENCE.RUNNING
   "DB442_MACHINE_RUN_OUT_ALARM_DECODING".UNIT_1.ALARM_RESET_LOCAL_SEQ_AUX.PULSES[3] := "DB1203_UNIT_1_STATION_1_CYCLE".SEQUENCE.RUNNING;
   IF #_w2 THEN
       "DB442_MACHINE_RUN_OUT_ALARM_DECODING".UNIT_1.ALARM_RESET_LOCAL_SEQ_AUX.STATION_1 := FALSE;
   END_IF;
END_REGION

REGION Network 16: RESET LOCAL SEQUENCES STATION 3
   RUNG wire#powerrail
      Contact( "M_ONE" )
      wire#w1
      P_Contact(operand := "DB442_MACHINE_RUN_OUT_ALARM_DECODING".UNIT_1.STATION_3.RHP_RO_ALARMS, bit := "DB442_MACHINE_RUN_OUT_ALARM_DECODING".UNIT_1.ALARM_RESET_LOCAL_SEQ_AUX.PULSES[4])
      S_Coil( "DB442_MACHINE_RUN_OUT_ALARM_DECODING".UNIT_1.ALARM_RESET_LOCAL_SEQ_AUX.STATION_3 )
   END_RUNG
   RUNG wire#w1
      N_Contact(operand := "DB1205_UNIT_1_STATION_3_CYCLE".SEQUENCE.RUNNING, bit := "DB442_MACHINE_RUN_OUT_ALARM_DECODING".UNIT_1.ALARM_RESET_LOCAL_SEQ_AUX.PULSES[5])
      wire#w2
      R_Coil( "DB442_MACHINE_RUN_OUT_ALARM_DECODING".UNIT_1.ALARM_RESET_LOCAL_SEQ_AUX.STATION_3 )
   END_RUNG
   RUNG wire#w1
      Contact( "DB2031_CYCLES_GENERAL".CALIBRATION_CYCLE.CYCLE_SELECTED )
      N_Contact(operand := "DB1235_UNIT_1_STATION_3_MEAS_CALIBRATION".SEQUENCE.RUNNING, bit := "DB442_MACHINE_RUN_OUT_ALARM_DECODING".UNIT_1.ALARM_RESET_LOCAL_SEQ_AUX.PULSES[8])
   END_RUNG wire#w2
   // the same network as SCL:
   #_w1 := "M_ONE" AND "DB442_MACHINE_RUN_OUT_ALARM_DECODING".UNIT_1.STATION_3.RHP_RO_ALARMS AND NOT "DB442_MACHINE_RUN_OUT_ALARM_DECODING".UNIT_1.ALARM_RESET_LOCAL_SEQ_AUX.PULSES[4];   // rising edge of "DB442_MACHINE_RUN_OUT_ALARM_DECODING".UNIT_1.STATION_3.RHP_RO_ALARMS
   "DB442_MACHINE_RUN_OUT_ALARM_DECODING".UNIT_1.ALARM_RESET_LOCAL_SEQ_AUX.PULSES[4] := "DB442_MACHINE_RUN_OUT_ALARM_DECODING".UNIT_1.STATION_3.RHP_RO_ALARMS;
   IF #_w1 THEN
       "DB442_MACHINE_RUN_OUT_ALARM_DECODING".UNIT_1.ALARM_RESET_LOCAL_SEQ_AUX.STATION_3 := TRUE;
   END_IF;
   #_w2 := "M_ONE" AND NOT "DB1205_UNIT_1_STATION_3_CYCLE".SEQUENCE.RUNNING AND "DB442_MACHINE_RUN_OUT_ALARM_DECODING".UNIT_1.ALARM_RESET_LOCAL_SEQ_AUX.PULSES[5];   // falling edge of "DB1205_UNIT_1_STATION_3_CYCLE".SEQUENCE.RUNNING
   "DB442_MACHINE_RUN_OUT_ALARM_DECODING".UNIT_1.ALARM_RESET_LOCAL_SEQ_AUX.PULSES[5] := "DB1205_UNIT_1_STATION_3_CYCLE".SEQUENCE.RUNNING;
   #_w3 := "M_ONE" AND "DB2031_CYCLES_GENERAL".CALIBRATION_CYCLE.CYCLE_SELECTED AND NOT "DB1235_UNIT_1_STATION_3_MEAS_CALIBRATION".SEQUENCE.RUNNING AND "DB442_MACHINE_RUN_OUT_ALARM_DECODING".UNIT_1.ALARM_RESET_LOCAL_SEQ_AUX.PULSES[8];   // falling edge of "DB1235_UNIT_1_STATION_3_MEAS_CALIBRATION".SEQUENCE.RUNNING
   "DB442_MACHINE_RUN_OUT_ALARM_DECODING".UNIT_1.ALARM_RESET_LOCAL_SEQ_AUX.PULSES[8] := "DB1235_UNIT_1_STATION_3_MEAS_CALIBRATION".SEQUENCE.RUNNING;
   IF #_w2 OR #_w3 THEN
       "DB442_MACHINE_RUN_OUT_ALARM_DECODING".UNIT_1.ALARM_RESET_LOCAL_SEQ_AUX.STATION_3 := FALSE;
   END_IF;
END_REGION

REGION Network 17: RESET LOCAL SEQUENCES STATION 4
   RUNG wire#powerrail
      Contact( "M_ONE" )
      wire#w1
      P_Contact(operand := "DB442_MACHINE_RUN_OUT_ALARM_DECODING".UNIT_1.STATION_4.RHP_RO_ALARMS, bit := "DB442_MACHINE_RUN_OUT_ALARM_DECODING".UNIT_1.ALARM_RESET_LOCAL_SEQ_AUX.PULSES[6])
      S_Coil( "DB442_MACHINE_RUN_OUT_ALARM_DECODING".UNIT_1.ALARM_RESET_LOCAL_SEQ_AUX.STATION_4 )
   END_RUNG
   RUNG wire#w1
      N_Contact(operand := "DB1206_UNIT_1_STATION_4_CYCLE".SEQUENCE.RUNNING, bit := "DB442_MACHINE_RUN_OUT_ALARM_DECODING".UNIT_1.ALARM_RESET_LOCAL_SEQ_AUX.PULSES[7])
      R_Coil( "DB442_MACHINE_RUN_OUT_ALARM_DECODING".UNIT_1.ALARM_RESET_LOCAL_SEQ_AUX.STATION_4 )
   END_RUNG
   // the same network as SCL:
   #_w1 := "M_ONE" AND "DB442_MACHINE_RUN_OUT_ALARM_DECODING".UNIT_1.STATION_4.RHP_RO_ALARMS AND NOT "DB442_MACHINE_RUN_OUT_ALARM_DECODING".UNIT_1.ALARM_RESET_LOCAL_SEQ_AUX.PULSES[6];   // rising edge of "DB442_MACHINE_RUN_OUT_ALARM_DECODING".UNIT_1.STATION_4.RHP_RO_ALARMS
   "DB442_MACHINE_RUN_OUT_ALARM_DECODING".UNIT_1.ALARM_RESET_LOCAL_SEQ_AUX.PULSES[6] := "DB442_MACHINE_RUN_OUT_ALARM_DECODING".UNIT_1.STATION_4.RHP_RO_ALARMS;
   IF #_w1 THEN
       "DB442_MACHINE_RUN_OUT_ALARM_DECODING".UNIT_1.ALARM_RESET_LOCAL_SEQ_AUX.STATION_4 := TRUE;
   END_IF;
   #_w2 := "M_ONE" AND NOT "DB1206_UNIT_1_STATION_4_CYCLE".SEQUENCE.RUNNING AND "DB442_MACHINE_RUN_OUT_ALARM_DECODING".UNIT_1.ALARM_RESET_LOCAL_SEQ_AUX.PULSES[7];   // falling edge of "DB1206_UNIT_1_STATION_4_CYCLE".SEQUENCE.RUNNING
   "DB442_MACHINE_RUN_OUT_ALARM_DECODING".UNIT_1.ALARM_RESET_LOCAL_SEQ_AUX.PULSES[7] := "DB1206_UNIT_1_STATION_4_CYCLE".SEQUENCE.RUNNING;
   IF #_w2 THEN
       "DB442_MACHINE_RUN_OUT_ALARM_DECODING".UNIT_1.ALARM_RESET_LOCAL_SEQ_AUX.STATION_4 := FALSE;
   END_IF;
END_REGION

REGION Network 18: <<<<<<<<<<<<<< RESET LOCAL SEQUENCES AUXILIAR UNIT 2 >>>>>>>>>>>>>>
END_REGION

REGION Network 19: RESET LOCAL SEQUENCES STATION 0
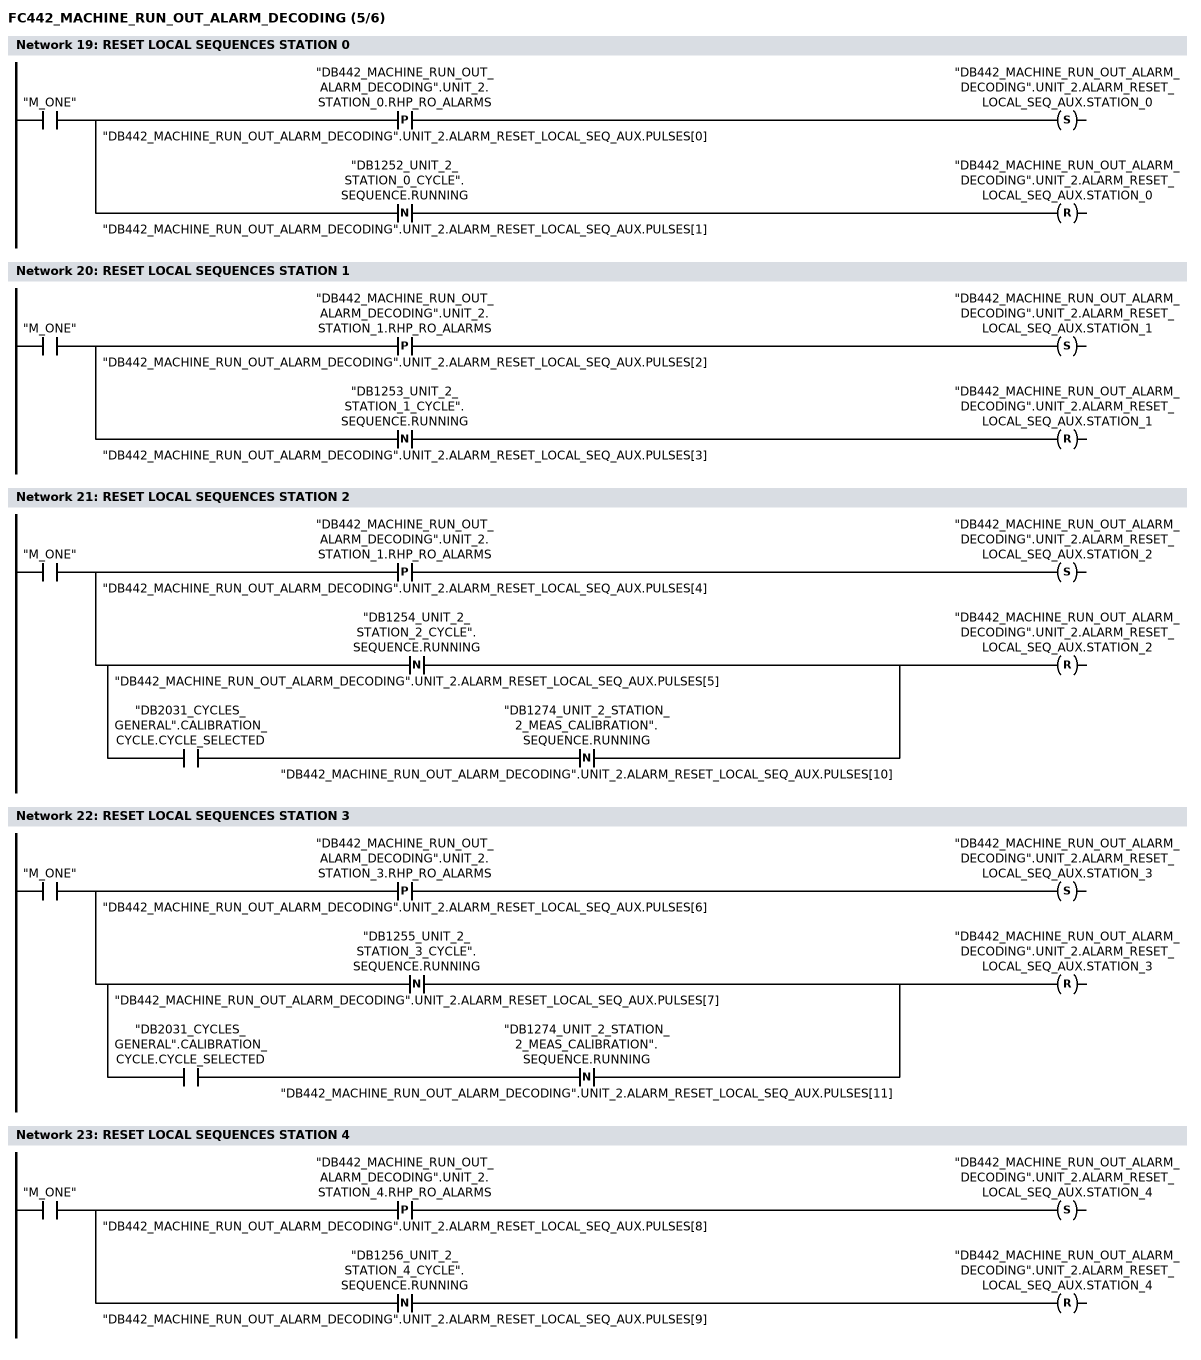
   RUNG wire#powerrail
      Contact( "M_ONE" )
      wire#w1
      P_Contact(operand := "DB442_MACHINE_RUN_OUT_ALARM_DECODING".UNIT_2.STATION_0.RHP_RO_ALARMS, bit := "DB442_MACHINE_RUN_OUT_ALARM_DECODING".UNIT_2.ALARM_RESET_LOCAL_SEQ_AUX.PULSES[0])
      S_Coil( "DB442_MACHINE_RUN_OUT_ALARM_DECODING".UNIT_2.ALARM_RESET_LOCAL_SEQ_AUX.STATION_0 )
   END_RUNG
   RUNG wire#w1
      N_Contact(operand := "DB1252_UNIT_2_STATION_0_CYCLE".SEQUENCE.RUNNING, bit := "DB442_MACHINE_RUN_OUT_ALARM_DECODING".UNIT_2.ALARM_RESET_LOCAL_SEQ_AUX.PULSES[1])
      R_Coil( "DB442_MACHINE_RUN_OUT_ALARM_DECODING".UNIT_2.ALARM_RESET_LOCAL_SEQ_AUX.STATION_0 )
   END_RUNG
   // the same network as SCL:
   #_w1 := "M_ONE" AND "DB442_MACHINE_RUN_OUT_ALARM_DECODING".UNIT_2.STATION_0.RHP_RO_ALARMS AND NOT "DB442_MACHINE_RUN_OUT_ALARM_DECODING".UNIT_2.ALARM_RESET_LOCAL_SEQ_AUX.PULSES[0];   // rising edge of "DB442_MACHINE_RUN_OUT_ALARM_DECODING".UNIT_2.STATION_0.RHP_RO_ALARMS
   "DB442_MACHINE_RUN_OUT_ALARM_DECODING".UNIT_2.ALARM_RESET_LOCAL_SEQ_AUX.PULSES[0] := "DB442_MACHINE_RUN_OUT_ALARM_DECODING".UNIT_2.STATION_0.RHP_RO_ALARMS;
   IF #_w1 THEN
       "DB442_MACHINE_RUN_OUT_ALARM_DECODING".UNIT_2.ALARM_RESET_LOCAL_SEQ_AUX.STATION_0 := TRUE;
   END_IF;
   #_w2 := "M_ONE" AND NOT "DB1252_UNIT_2_STATION_0_CYCLE".SEQUENCE.RUNNING AND "DB442_MACHINE_RUN_OUT_ALARM_DECODING".UNIT_2.ALARM_RESET_LOCAL_SEQ_AUX.PULSES[1];   // falling edge of "DB1252_UNIT_2_STATION_0_CYCLE".SEQUENCE.RUNNING
   "DB442_MACHINE_RUN_OUT_ALARM_DECODING".UNIT_2.ALARM_RESET_LOCAL_SEQ_AUX.PULSES[1] := "DB1252_UNIT_2_STATION_0_CYCLE".SEQUENCE.RUNNING;
   IF #_w2 THEN
       "DB442_MACHINE_RUN_OUT_ALARM_DECODING".UNIT_2.ALARM_RESET_LOCAL_SEQ_AUX.STATION_0 := FALSE;
   END_IF;
END_REGION

REGION Network 20: RESET LOCAL SEQUENCES STATION 1
   RUNG wire#powerrail
      Contact( "M_ONE" )
      wire#w1
      P_Contact(operand := "DB442_MACHINE_RUN_OUT_ALARM_DECODING".UNIT_2.STATION_1.RHP_RO_ALARMS, bit := "DB442_MACHINE_RUN_OUT_ALARM_DECODING".UNIT_2.ALARM_RESET_LOCAL_SEQ_AUX.PULSES[2])
      S_Coil( "DB442_MACHINE_RUN_OUT_ALARM_DECODING".UNIT_2.ALARM_RESET_LOCAL_SEQ_AUX.STATION_1 )
   END_RUNG
   RUNG wire#w1
      N_Contact(operand := "DB1253_UNIT_2_STATION_1_CYCLE".SEQUENCE.RUNNING, bit := "DB442_MACHINE_RUN_OUT_ALARM_DECODING".UNIT_2.ALARM_RESET_LOCAL_SEQ_AUX.PULSES[3])
      R_Coil( "DB442_MACHINE_RUN_OUT_ALARM_DECODING".UNIT_2.ALARM_RESET_LOCAL_SEQ_AUX.STATION_1 )
   END_RUNG
   // the same network as SCL:
   #_w1 := "M_ONE" AND "DB442_MACHINE_RUN_OUT_ALARM_DECODING".UNIT_2.STATION_1.RHP_RO_ALARMS AND NOT "DB442_MACHINE_RUN_OUT_ALARM_DECODING".UNIT_2.ALARM_RESET_LOCAL_SEQ_AUX.PULSES[2];   // rising edge of "DB442_MACHINE_RUN_OUT_ALARM_DECODING".UNIT_2.STATION_1.RHP_RO_ALARMS
   "DB442_MACHINE_RUN_OUT_ALARM_DECODING".UNIT_2.ALARM_RESET_LOCAL_SEQ_AUX.PULSES[2] := "DB442_MACHINE_RUN_OUT_ALARM_DECODING".UNIT_2.STATION_1.RHP_RO_ALARMS;
   IF #_w1 THEN
       "DB442_MACHINE_RUN_OUT_ALARM_DECODING".UNIT_2.ALARM_RESET_LOCAL_SEQ_AUX.STATION_1 := TRUE;
   END_IF;
   #_w2 := "M_ONE" AND NOT "DB1253_UNIT_2_STATION_1_CYCLE".SEQUENCE.RUNNING AND "DB442_MACHINE_RUN_OUT_ALARM_DECODING".UNIT_2.ALARM_RESET_LOCAL_SEQ_AUX.PULSES[3];   // falling edge of "DB1253_UNIT_2_STATION_1_CYCLE".SEQUENCE.RUNNING
   "DB442_MACHINE_RUN_OUT_ALARM_DECODING".UNIT_2.ALARM_RESET_LOCAL_SEQ_AUX.PULSES[3] := "DB1253_UNIT_2_STATION_1_CYCLE".SEQUENCE.RUNNING;
   IF #_w2 THEN
       "DB442_MACHINE_RUN_OUT_ALARM_DECODING".UNIT_2.ALARM_RESET_LOCAL_SEQ_AUX.STATION_1 := FALSE;
   END_IF;
END_REGION

REGION Network 21: RESET LOCAL SEQUENCES STATION 2
   RUNG wire#powerrail
      Contact( "M_ONE" )
      wire#w1
      P_Contact(operand := "DB442_MACHINE_RUN_OUT_ALARM_DECODING".UNIT_2.STATION_1.RHP_RO_ALARMS, bit := "DB442_MACHINE_RUN_OUT_ALARM_DECODING".UNIT_2.ALARM_RESET_LOCAL_SEQ_AUX.PULSES[4])
      S_Coil( "DB442_MACHINE_RUN_OUT_ALARM_DECODING".UNIT_2.ALARM_RESET_LOCAL_SEQ_AUX.STATION_2 )
   END_RUNG
   RUNG wire#w1
      N_Contact(operand := "DB1254_UNIT_2_STATION_2_CYCLE".SEQUENCE.RUNNING, bit := "DB442_MACHINE_RUN_OUT_ALARM_DECODING".UNIT_2.ALARM_RESET_LOCAL_SEQ_AUX.PULSES[5])
      wire#w2
      R_Coil( "DB442_MACHINE_RUN_OUT_ALARM_DECODING".UNIT_2.ALARM_RESET_LOCAL_SEQ_AUX.STATION_2 )
   END_RUNG
   RUNG wire#w1
      Contact( "DB2031_CYCLES_GENERAL".CALIBRATION_CYCLE.CYCLE_SELECTED )
      N_Contact(operand := "DB1274_UNIT_2_STATION_2_MEAS_CALIBRATION".SEQUENCE.RUNNING, bit := "DB442_MACHINE_RUN_OUT_ALARM_DECODING".UNIT_2.ALARM_RESET_LOCAL_SEQ_AUX.PULSES[10])
   END_RUNG wire#w2
   // the same network as SCL:
   #_w1 := "M_ONE" AND "DB442_MACHINE_RUN_OUT_ALARM_DECODING".UNIT_2.STATION_1.RHP_RO_ALARMS AND NOT "DB442_MACHINE_RUN_OUT_ALARM_DECODING".UNIT_2.ALARM_RESET_LOCAL_SEQ_AUX.PULSES[4];   // rising edge of "DB442_MACHINE_RUN_OUT_ALARM_DECODING".UNIT_2.STATION_1.RHP_RO_ALARMS
   "DB442_MACHINE_RUN_OUT_ALARM_DECODING".UNIT_2.ALARM_RESET_LOCAL_SEQ_AUX.PULSES[4] := "DB442_MACHINE_RUN_OUT_ALARM_DECODING".UNIT_2.STATION_1.RHP_RO_ALARMS;
   IF #_w1 THEN
       "DB442_MACHINE_RUN_OUT_ALARM_DECODING".UNIT_2.ALARM_RESET_LOCAL_SEQ_AUX.STATION_2 := TRUE;
   END_IF;
   #_w2 := "M_ONE" AND NOT "DB1254_UNIT_2_STATION_2_CYCLE".SEQUENCE.RUNNING AND "DB442_MACHINE_RUN_OUT_ALARM_DECODING".UNIT_2.ALARM_RESET_LOCAL_SEQ_AUX.PULSES[5];   // falling edge of "DB1254_UNIT_2_STATION_2_CYCLE".SEQUENCE.RUNNING
   "DB442_MACHINE_RUN_OUT_ALARM_DECODING".UNIT_2.ALARM_RESET_LOCAL_SEQ_AUX.PULSES[5] := "DB1254_UNIT_2_STATION_2_CYCLE".SEQUENCE.RUNNING;
   #_w3 := "M_ONE" AND "DB2031_CYCLES_GENERAL".CALIBRATION_CYCLE.CYCLE_SELECTED AND NOT "DB1274_UNIT_2_STATION_2_MEAS_CALIBRATION".SEQUENCE.RUNNING AND "DB442_MACHINE_RUN_OUT_ALARM_DECODING".UNIT_2.ALARM_RESET_LOCAL_SEQ_AUX.PULSES[10];   // falling edge of "DB1274_UNIT_2_STATION_2_MEAS_CALIBRATION".SEQUENCE.RUNNING
   "DB442_MACHINE_RUN_OUT_ALARM_DECODING".UNIT_2.ALARM_RESET_LOCAL_SEQ_AUX.PULSES[10] := "DB1274_UNIT_2_STATION_2_MEAS_CALIBRATION".SEQUENCE.RUNNING;
   IF #_w2 OR #_w3 THEN
       "DB442_MACHINE_RUN_OUT_ALARM_DECODING".UNIT_2.ALARM_RESET_LOCAL_SEQ_AUX.STATION_2 := FALSE;
   END_IF;
END_REGION

REGION Network 22: RESET LOCAL SEQUENCES STATION 3
   RUNG wire#powerrail
      Contact( "M_ONE" )
      wire#w1
      P_Contact(operand := "DB442_MACHINE_RUN_OUT_ALARM_DECODING".UNIT_2.STATION_3.RHP_RO_ALARMS, bit := "DB442_MACHINE_RUN_OUT_ALARM_DECODING".UNIT_2.ALARM_RESET_LOCAL_SEQ_AUX.PULSES[6])
      S_Coil( "DB442_MACHINE_RUN_OUT_ALARM_DECODING".UNIT_2.ALARM_RESET_LOCAL_SEQ_AUX.STATION_3 )
   END_RUNG
   RUNG wire#w1
      N_Contact(operand := "DB1255_UNIT_2_STATION_3_CYCLE".SEQUENCE.RUNNING, bit := "DB442_MACHINE_RUN_OUT_ALARM_DECODING".UNIT_2.ALARM_RESET_LOCAL_SEQ_AUX.PULSES[7])
      wire#w2
      R_Coil( "DB442_MACHINE_RUN_OUT_ALARM_DECODING".UNIT_2.ALARM_RESET_LOCAL_SEQ_AUX.STATION_3 )
   END_RUNG
   RUNG wire#w1
      Contact( "DB2031_CYCLES_GENERAL".CALIBRATION_CYCLE.CYCLE_SELECTED )
      N_Contact(operand := "DB1274_UNIT_2_STATION_2_MEAS_CALIBRATION".SEQUENCE.RUNNING, bit := "DB442_MACHINE_RUN_OUT_ALARM_DECODING".UNIT_2.ALARM_RESET_LOCAL_SEQ_AUX.PULSES[11])
   END_RUNG wire#w2
   // the same network as SCL:
   #_w1 := "M_ONE" AND "DB442_MACHINE_RUN_OUT_ALARM_DECODING".UNIT_2.STATION_3.RHP_RO_ALARMS AND NOT "DB442_MACHINE_RUN_OUT_ALARM_DECODING".UNIT_2.ALARM_RESET_LOCAL_SEQ_AUX.PULSES[6];   // rising edge of "DB442_MACHINE_RUN_OUT_ALARM_DECODING".UNIT_2.STATION_3.RHP_RO_ALARMS
   "DB442_MACHINE_RUN_OUT_ALARM_DECODING".UNIT_2.ALARM_RESET_LOCAL_SEQ_AUX.PULSES[6] := "DB442_MACHINE_RUN_OUT_ALARM_DECODING".UNIT_2.STATION_3.RHP_RO_ALARMS;
   IF #_w1 THEN
       "DB442_MACHINE_RUN_OUT_ALARM_DECODING".UNIT_2.ALARM_RESET_LOCAL_SEQ_AUX.STATION_3 := TRUE;
   END_IF;
   #_w2 := "M_ONE" AND NOT "DB1255_UNIT_2_STATION_3_CYCLE".SEQUENCE.RUNNING AND "DB442_MACHINE_RUN_OUT_ALARM_DECODING".UNIT_2.ALARM_RESET_LOCAL_SEQ_AUX.PULSES[7];   // falling edge of "DB1255_UNIT_2_STATION_3_CYCLE".SEQUENCE.RUNNING
   "DB442_MACHINE_RUN_OUT_ALARM_DECODING".UNIT_2.ALARM_RESET_LOCAL_SEQ_AUX.PULSES[7] := "DB1255_UNIT_2_STATION_3_CYCLE".SEQUENCE.RUNNING;
   #_w3 := "M_ONE" AND "DB2031_CYCLES_GENERAL".CALIBRATION_CYCLE.CYCLE_SELECTED AND NOT "DB1274_UNIT_2_STATION_2_MEAS_CALIBRATION".SEQUENCE.RUNNING AND "DB442_MACHINE_RUN_OUT_ALARM_DECODING".UNIT_2.ALARM_RESET_LOCAL_SEQ_AUX.PULSES[11];   // falling edge of "DB1274_UNIT_2_STATION_2_MEAS_CALIBRATION".SEQUENCE.RUNNING
   "DB442_MACHINE_RUN_OUT_ALARM_DECODING".UNIT_2.ALARM_RESET_LOCAL_SEQ_AUX.PULSES[11] := "DB1274_UNIT_2_STATION_2_MEAS_CALIBRATION".SEQUENCE.RUNNING;
   IF #_w2 OR #_w3 THEN
       "DB442_MACHINE_RUN_OUT_ALARM_DECODING".UNIT_2.ALARM_RESET_LOCAL_SEQ_AUX.STATION_3 := FALSE;
   END_IF;
END_REGION

REGION Network 23: RESET LOCAL SEQUENCES STATION 4
   RUNG wire#powerrail
      Contact( "M_ONE" )
      wire#w1
      P_Contact(operand := "DB442_MACHINE_RUN_OUT_ALARM_DECODING".UNIT_2.STATION_4.RHP_RO_ALARMS, bit := "DB442_MACHINE_RUN_OUT_ALARM_DECODING".UNIT_2.ALARM_RESET_LOCAL_SEQ_AUX.PULSES[8])
      S_Coil( "DB442_MACHINE_RUN_OUT_ALARM_DECODING".UNIT_2.ALARM_RESET_LOCAL_SEQ_AUX.STATION_4 )
   END_RUNG
   RUNG wire#w1
      N_Contact(operand := "DB1256_UNIT_2_STATION_4_CYCLE".SEQUENCE.RUNNING, bit := "DB442_MACHINE_RUN_OUT_ALARM_DECODING".UNIT_2.ALARM_RESET_LOCAL_SEQ_AUX.PULSES[9])
      R_Coil( "DB442_MACHINE_RUN_OUT_ALARM_DECODING".UNIT_2.ALARM_RESET_LOCAL_SEQ_AUX.STATION_4 )
   END_RUNG
   // the same network as SCL:
   #_w1 := "M_ONE" AND "DB442_MACHINE_RUN_OUT_ALARM_DECODING".UNIT_2.STATION_4.RHP_RO_ALARMS AND NOT "DB442_MACHINE_RUN_OUT_ALARM_DECODING".UNIT_2.ALARM_RESET_LOCAL_SEQ_AUX.PULSES[8];   // rising edge of "DB442_MACHINE_RUN_OUT_ALARM_DECODING".UNIT_2.STATION_4.RHP_RO_ALARMS
   "DB442_MACHINE_RUN_OUT_ALARM_DECODING".UNIT_2.ALARM_RESET_LOCAL_SEQ_AUX.PULSES[8] := "DB442_MACHINE_RUN_OUT_ALARM_DECODING".UNIT_2.STATION_4.RHP_RO_ALARMS;
   IF #_w1 THEN
       "DB442_MACHINE_RUN_OUT_ALARM_DECODING".UNIT_2.ALARM_RESET_LOCAL_SEQ_AUX.STATION_4 := TRUE;
   END_IF;
   #_w2 := "M_ONE" AND NOT "DB1256_UNIT_2_STATION_4_CYCLE".SEQUENCE.RUNNING AND "DB442_MACHINE_RUN_OUT_ALARM_DECODING".UNIT_2.ALARM_RESET_LOCAL_SEQ_AUX.PULSES[9];   // falling edge of "DB1256_UNIT_2_STATION_4_CYCLE".SEQUENCE.RUNNING
   "DB442_MACHINE_RUN_OUT_ALARM_DECODING".UNIT_2.ALARM_RESET_LOCAL_SEQ_AUX.PULSES[9] := "DB1256_UNIT_2_STATION_4_CYCLE".SEQUENCE.RUNNING;
   IF #_w2 THEN
       "DB442_MACHINE_RUN_OUT_ALARM_DECODING".UNIT_2.ALARM_RESET_LOCAL_SEQ_AUX.STATION_4 := FALSE;
   END_IF;
END_REGION

REGION Network 24: <<<<<<<<<<<<<< RESET LOCAL SEQUENCES AUXILIAR UNIT 3 >>>>>>>>>>>>>>
END_REGION

REGION Network 25: RESET LOCAL SEQUENCES CONTROL STATION
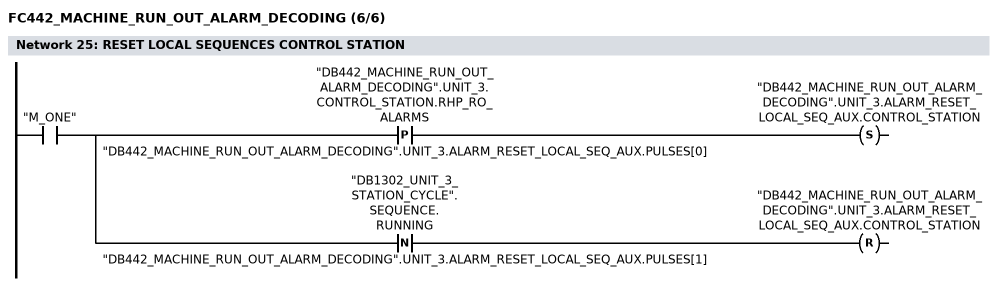
   RUNG wire#powerrail
      Contact( "M_ONE" )
      wire#w1
      P_Contact(operand := "DB442_MACHINE_RUN_OUT_ALARM_DECODING".UNIT_3.CONTROL_STATION.RHP_RO_ALARMS, bit := "DB442_MACHINE_RUN_OUT_ALARM_DECODING".UNIT_3.ALARM_RESET_LOCAL_SEQ_AUX.PULSES[0])
      S_Coil( "DB442_MACHINE_RUN_OUT_ALARM_DECODING".UNIT_3.ALARM_RESET_LOCAL_SEQ_AUX.CONTROL_STATION )
   END_RUNG
   RUNG wire#w1
      N_Contact(operand := "DB1302_UNIT_3_STATION_CYCLE".SEQUENCE.RUNNING, bit := "DB442_MACHINE_RUN_OUT_ALARM_DECODING".UNIT_3.ALARM_RESET_LOCAL_SEQ_AUX.PULSES[1])
      R_Coil( "DB442_MACHINE_RUN_OUT_ALARM_DECODING".UNIT_3.ALARM_RESET_LOCAL_SEQ_AUX.CONTROL_STATION )
   END_RUNG
   // the same network as SCL:
   #_w1 := "M_ONE" AND "DB442_MACHINE_RUN_OUT_ALARM_DECODING".UNIT_3.CONTROL_STATION.RHP_RO_ALARMS AND NOT "DB442_MACHINE_RUN_OUT_ALARM_DECODING".UNIT_3.ALARM_RESET_LOCAL_SEQ_AUX.PULSES[0];   // rising edge of "DB442_MACHINE_RUN_OUT_ALARM_DECODING".UNIT_3.CONTROL_STATION.RHP_RO_ALARMS
   "DB442_MACHINE_RUN_OUT_ALARM_DECODING".UNIT_3.ALARM_RESET_LOCAL_SEQ_AUX.PULSES[0] := "DB442_MACHINE_RUN_OUT_ALARM_DECODING".UNIT_3.CONTROL_STATION.RHP_RO_ALARMS;
   IF #_w1 THEN
       "DB442_MACHINE_RUN_OUT_ALARM_DECODING".UNIT_3.ALARM_RESET_LOCAL_SEQ_AUX.CONTROL_STATION := TRUE;
   END_IF;
   #_w2 := "M_ONE" AND NOT "DB1302_UNIT_3_STATION_CYCLE".SEQUENCE.RUNNING AND "DB442_MACHINE_RUN_OUT_ALARM_DECODING".UNIT_3.ALARM_RESET_LOCAL_SEQ_AUX.PULSES[1];   // falling edge of "DB1302_UNIT_3_STATION_CYCLE".SEQUENCE.RUNNING
   "DB442_MACHINE_RUN_OUT_ALARM_DECODING".UNIT_3.ALARM_RESET_LOCAL_SEQ_AUX.PULSES[1] := "DB1302_UNIT_3_STATION_CYCLE".SEQUENCE.RUNNING;
   IF #_w2 THEN
       "DB442_MACHINE_RUN_OUT_ALARM_DECODING".UNIT_3.ALARM_RESET_LOCAL_SEQ_AUX.CONTROL_STATION := FALSE;
   END_IF;
END_REGION
END_FUNCTION
